VAR
    
END_VAR


// Koffieapparaat aanzetten zodra gebruiker wakker is
IF GVL.g_bWakker THEN
    GVL.g_KoffieZetten(IN := TRUE, PT := T#10S);  // Koffie loopt voor 10 seconden
ELSE
    GVL.g_KoffieZetten(IN := FALSE);
END_IF

// Koffie is klaar zodra de timer klaar is
IF GVL.g_KoffieZetten.Q THEN
    GVL.g_bKoffieKlaar := TRUE;
END_IF

(* stored: Version 1.1.0.1, ProductVersion 3.1.4024.15
   POU TaskKoffieZetten: Id {3747bf79-b671-48c5-b96f-b14694d16c67}, SpecialFunc None *)
